INTERFACE IAssertionMessageList

METHOD AddMessage : BOOL
VAR_INPUT
    Message : T_MaxString;
END_VAR
END_METHOD

METHOD Clear
VAR_INPUT
END_VAR
END_METHOD

END_INTERFACE

(* stored: Version 1.1.0.1, ProductVersion 3.1.4024.4
   Itf IAssertionMessageList: Id {4656d820-d7df-49e3-8843-f40bfefe0cbb}
   Method AddMessage: Id {6b8d80e4-67be-4a8a-b966-e5307dbe0a90}
   Method Clear: Id {f1f39b29-d68a-4218-bc7c-cb02814d7b61} *)
